// TwinCAT 3 PLC project LF_System_PLC
// ProgramVersion: 3.1.4026.20
// CompilerDefines: VISU_USEPROPERTYINFO
// libraries:
//   Tc2_Standard, * (Beckhoff Automation GmbH)
//   Tc2_System, * (Beckhoff Automation GmbH)
//   VisuSymbols, 4.5.0.0 (System)
// project tree:
//   / GlobalTextList.TcGTLO, PlcTask.TcTTO, Visualization Manager.TcVMO (not stored)
//   POUs/Extruder/ FB_System_FlaschenFullstand.TcPOU, FB_System_Fullstand.TcPOU
//   POUs/ FB_System_CNV.TcPOU (not stored), MAIN.TcPOU
//   POUs/Vereinzelung/ FB_SpeicherRohr.TcPOU, FB_System_Vereinzelung.TcPOU
//   VISUs/ Visualization.TcVIS
// (motion and I/O tree: see PLC project tempmodel)
// real-time tasks:
//   TASK PlcTask: cycle T#10ms, priority 21, ADS port 350
//   TASK PlcTask1: cycle T#10ms, priority 22, ADS port 351
//   TASK PlcTask2: cycle T#10ms, priority 20, ADS port 352
// variable links:
//   LF_System_PLC/LF_System_PLC Instance <-> NC-Task 1 SAF/Axes/BandAchse
//     PlcTask Inputs/MAIN.fIN_CnvPos <-> Outputs/ToPlc/ActPos
//   LF_System_PLC/LF_System_PLC Instance <-> PLC/PLC Instance
//     PlcTask Inputs/MAIN.bIn_LedGreen <-> PlcTask Outputs/IFC_HW.bAmpelGrun
//     PlcTask Inputs/MAIN.bIn_LedRot <-> PlcTask Outputs/IFC_HW.bAmpelRot
//     PlcTask Inputs/MAIN.bIn_LedYellow <-> PlcTask Outputs/IFC_HW.bAmpelGelb
//     PlcTask Inputs/MAIN.bIn_Schleuse1_L1 <-> PlcTask Outputs/IFC_HW.bR1AKT1
//     PlcTask Inputs/MAIN.bIn_Schleuse1_L2 <-> PlcTask Outputs/IFC_HW.bR2AKT1
//     PlcTask Inputs/MAIN.bIn_Schleuse2_L1 <-> PlcTask Outputs/IFC_HW.bR1AKT2
//     PlcTask Inputs/MAIN.bIn_Schleuse2_L2 <-> PlcTask Outputs/IFC_HW.bR2AKT2
//     PlcTask Outputs/MAIN.bEnable <-> PlcTask Inputs/IFC_HW.bEnable
//     PlcTask Outputs/MAIN.bExecute <-> PlcTask Inputs/IFC_HW.bExecute
//     PlcTask Outputs/MAIN.bOut_VereinzelungNS1 <-> PlcTask Inputs/IFC_HW.bEinzelSens3
//     PlcTask Outputs/MAIN.bOut_VereinzelungNS2 <-> PlcTask Inputs/IFC_HW.bEinzelSens2
//     PlcTask Outputs/MAIN.bOut_VereinzelungNS3 <-> PlcTask Inputs/IFC_HW.bEinzelSens1

CONFIGURATION LF_System_PLC
    RESOURCE PLC ON TwinCAT3
        TASK PlcTask(INTERVAL := T#10ms, PRIORITY := 22);
        PROGRAM MAIN WITH PlcTask : MAIN;
    END_RESOURCE
END_CONFIGURATION

// ---- POUs/MAIN.TcPOU
PROGRAM MAIN
VAR
// Systemeingangssignale (Stellsignale für Aktoren)
	bEnable AT%Q* : BOOL;
	bExecute AT%Q* : BOOL;
	// Status Lampe
	bIn_LedRot 		AT%I* : BOOL;
	bIn_LedYellow 	AT%I* : BOOL;
	bIn_LedGreen 	AT%I* : BOOL;
	// Vereinzelung 
	bIn_Schleuse1_L1 AT%I* : BOOL; // + Öffnen - Schließen
	bIn_Schleuse1_L2 AT%I* : BOOL; // + Schließen - Öffnen
	bIn_Schleuse2_L1 AT%I* : BOOL; // + Öffnen - Schließen
	bIn_Schleuse2_L2 AT%I* : BOOL; // + Schließen - Öffnen
	// Förderband
	fIN_CnvPos AT%I* : LREAL;
	bIN_Stopper1 AT%I* : BOOL;
	bIN_Stopper2 AT%I* : BOOL;
	bIN_Stopper3 AT%I* : BOOL;
	// Extruder
	fIN_ExtPos1 AT%I* : LREAL;
	fIN_ExtPos2 AT%I* : LREAL;
	fIN_ExtPos3 AT%I* : LREAL;
	
// Systemausgangssignale (Sensorsignale)
	//Vereinzelung
	bOut_VereinzelungNS1 AT%Q* : BOOL; // Flasche am Kopf
	bOut_VereinzelungNS2 AT%Q* : BOOL; // Flasche im Speicher
	bOut_VereinzelungNS3 AT%Q* : BOOL; // Flasche in Kammer
	//Förderband
	bOUT_CnvNS1 AT%Q* : BOOL;
	bOUT_CnvNS2 AT%Q* : BOOL;
	bOUT_CnvNS3 AT%Q* : BOOL;
	bOUT_CnvNS4 AT%Q* : BOOL;
	// Füllstandssensoren
	iOut_USS1 AT%Q* : UINT;
	iOut_USS2 AT%Q* : UINT;
	iOut_USS3 AT%Q* : UINT;
	
// System FB
	fbVereinzelung : FB_System_Vereinzelung;	
	fbCNV : FB_System_CNV;
	fbExt1 : FB_System_Fullstand;
	fbExt2 : FB_System_Fullstand;
	fbExt3 : FB_System_Fullstand;
	fbBottleLevel : FB_System_FlaschenFullstand;
	
// Hilfsvariablen
	bRefill1 : BOOL;
	bRefill2 : BOOL;
	bRefill3 : BOOL;
	bBottleDropped : BOOL;
	bBottleLeft : BOOL;
END_VAR

fbVereinzelung(
	bS1L1:= bIn_Schleuse1_L1, 
	bS1L2:= bIn_Schleuse1_L2, 
	bS2L1:= bIn_Schleuse2_L1, 
	bS2L2:= bIn_Schleuse2_L2,
	bNS1=> bOut_VereinzelungNS1, 
	bNS2=> bOut_VereinzelungNS2, 
	bNS3=> bOut_VereinzelungNS3,
	bBottleDropped => bBottleDropped);
	
fbCNV(
	fPos:= fIN_CnvPos, 
	bStopper1:= bIN_Stopper1, 
	bStopper2:= bIN_Stopper2, 
	bStopper3:= bIN_Stopper3, 
	bBottleDropped := bBottleDropped , 
	bNS1=> bOut_CnvNS1 , 
	bNS2=> bOut_CnvNS2 , 
	bNS3=> bOut_CnvNS3 , 
	bNS4=> bOut_CnvNS4,
	bBottleLeft => bBottleLeft);
	
fbExt1(bRefill:=bRefill1 , fPosExt:= fIN_ExtPos1, iOut=> iOut_USS1 );
fbExt2(bRefill:=bRefill2 , fPosExt:= fIN_ExtPos2, iOut=> iOut_USS2 );
fbExt3(bRefill:=bRefill3 , fPosExt:= fIN_ExtPos3, iOut=> iOut_USS3 );

fbBottleLevel(rFilling1 := fIN_ExtPos1, rFilling2 := fIN_ExtPos2 ,rFilling3 := fIN_ExtPos3,Reset:= bBottleLeft );

END_PROGRAM

// ---- POUs/Vereinzelung/FB_System_Vereinzelung.TcPOU
FUNCTION_BLOCK FB_System_Vereinzelung
VAR_INPUT
	bS1L1 : BOOL; // + Öffnen - Schließen
	bS1L2 : BOOL; // + Schließen - Öffnen
	bS2L1 : BOOL; // + Öffnen - Schließen
	bS2L2 : BOOL; // + Schließen - Öffnen
END_VAR
VAR_OUTPUT
	bNS1 : BOOL; // Flasche am Kopf
	bNS2 : BOOL; // Flasche im Speicher
	bNS3 : BOOL; // Flasche in Kammer
	bBottleDropped : BOOL;
END_VAR
VAR
	bS1open : BOOL;
	bS2open : BOOL;
	TimerS1 : Ton; // Schleusenbewegung (Schleuse1)
	TimerS2 : Ton; // Schleusenbewegung (Schleuse2)
	fbSpeicherRohr : FB_SpeicherRohr;
	nCaseS1 : UINT := 0;
	nCaseS2 : UINT := 0;
	bBefullen : BOOL;
	S1pos : INT;
	S2pos : INT;
END_VAR

TimerS1(PT := T#0.3S);
TimerS2(PT := T#0.3S);
fbSpeicherRohr(bFlascheBefullen:= bBefullen, bFlascheAuswurf := bS1open, bKammer := bNS3, bAuswurf => , aSpeicher => );

// Sensor in Speicher
bNS2 := fbSpeicherRohr.aSpeicher[0];
// Sensor in Kammer
IF fbSpeicherRohr.bAuswurf AND NOT bS2open THEN
	bNS3 := TRUE;
ELSIF bS2Open THEN
	bNS3 := FALSE;
END_IF

CASE nCaseS1 OF // Zustand S1
	0: // Schleuse geschlossen
	bS1open := FALSE;
	IF bS1L1 AND NOT bS1L2 THEN
		nCaseS1 := 1; // obere Schleuse öffnen
	END_IF
//------------------------------------------------	
	1: // obere Schleuse öffnen
	TimerS1.IN := TRUE;
	IF NOT bS1open THEN
		S1pos := S1pos - 1;
	END_IF
	IF TimerS1.Q THEN
		bS1open := TRUE;
	END_IF
	IF NOT bS1L1 AND bS1L2 THEN
		nCaseS1 := 2; // obere Schleuse schließen
		TimerS1.IN := FALSE;
	END_IF
//------------------------------------------------
	2: //obere Schleuse schließen
	TimerS1.IN := TRUE;
	IF bS1open THEN
		S1pos := S1pos + 1;
	END_IF
	IF timerS1.Q THEN
		bS1open := FALSE;
	END_IF
	IF bS1L1 AND NOT bS1L2 THEN
		nCaseS1 := 1; // obere Schleuse schließen
		TimerS1.IN := FALSE;
	END_IF
END_CASE

CASE nCaseS2 OF // Zustand S2
	0: // Schleuse geschlossen
	bS2open := FALSE;
	IF bS2L1 AND NOT bS2L2 THEN
		nCaseS2 := 1; // obere Schleuse öffnen
	END_IF
//------------------------------------------------	
	1: // untere Schleuse öffnen
	TimerS2.IN := TRUE;
	IF NOT bS2open THEN
		S2pos := S2pos - 1;
	END_IF
	IF TimerS2.Q THEN
		bS2open := TRUE;
	END_IF
	IF bS2open AND bNS3 THEN
		bBottleDropped := TRUE;
	END_IF
	IF NOT bS2L1 AND bS2L2 THEN
		nCaseS2 := 2; // untere Schleuse schließen
		TimerS2.IN := FALSE;
	END_IF
//------------------------------------------------
	2: //untere Schleuse schließen
	TimerS2.IN := TRUE;
	IF bS2open THEN
		S2pos := S2pos + 1;
	END_IF
	IF timerS2.Q THEN
		bS2open := FALSE;
		bBottleDropped := FALSE;
	END_IF
	IF bS2L1 AND NOT bS2L2 THEN
		nCaseS2 := 1; // untere Schleuse schließen
		TimerS2.IN := FALSE;
	END_IF
END_CASE

END_FUNCTION_BLOCK

// ---- POUs/Vereinzelung/FB_SpeicherRohr.TcPOU
FUNCTION_BLOCK FB_SpeicherRohr
VAR_INPUT
	bFlascheBefullen : BOOL; // Flasche soll in Speicher gelegt werden
	bFlascheAuswurf : BOOL; // Flasche soll in Kammer fallen
	bKammer : Bool;
END_VAR
VAR_OUTPUT
	bAuswurf : BOOL; // Flasche wurde ausgeworfen
	aSpeicher : ARRAY[0..3] OF BOOL := [TRUE,TRUE,TRUE,FALSE];
END_VAR
VAR
	rTrigBefullen : R_Trig;
	rTrigAuswurf : R_Trig;
	i : INT;
END_VAR

rTrigBefullen(CLK := bFlascheBefullen);
rTrigAuswurf(CLK := bFlascheAuswurf);

// Flaschenspeicher befüllen
IF rTrigBefullen.q AND NOT aSpeicher[3] THEN
	FOR i := 0 TO 3 DO
		IF NOT aSpeicher[i] THEN
			aSpeicher[i] := TRUE;
			EXIT;
		END_IF
	END_FOR
ELSIF rTrigBefullen.Q AND NOT aSpeicher[0] AND bFlascheAuswurf AND NOT bKammer THEN
	aSpeicher[0] := FALSE; 
	aSpeicher[1] := FALSE;
	aSpeicher[2] := FALSE;
	aSpeicher[3] := FALSE;
	bAuswurf := TRUE;
END_IF

IF rTrigAuswurf.q AND aSpeicher[0] THEN
	FOR i := 3 TO 0 BY -1 DO
		IF aSpeicher[i] THEN
			aSpeicher[i] := FALSE;
			EXIT;
		END_IF
	END_FOR
	bAuswurf := TRUE;
ELSE
	bAuswurf := FALSE; // Keine Flasche in Speicher
END_IF

END_FUNCTION_BLOCK

// ---- POUs/Extruder/FB_System_Fullstand.TcPOU
FUNCTION_BLOCK FB_System_Fullstand
VAR_INPUT
	bRefill : BOOL;
	fPosExt : LREAL;
END_VAR
VAR_OUTPUT
	iOut : UINT; // Fullstandssignal
END_VAR
VAR
	rPcntFillLevel : LREAL := 50.0; // Fullstand in Prozent
	iFillLevel : UINT;
	fPosExtAlt : LREAL;
	NotMoving : Bool;
END_VAR


// Auffüllen
IF bRefill THEN
	rPcntFillLevel := 100.0;
END_IF
// Füllstandsänderung durch Extruderbewegung
IF NOT notMoving THEN
	rPcntFillLevel := rPcntFillLevel - (fPosExt-fPosExtAlt)/360*0.5; // Füllstand - Grad/Umdrehung * 0,5% pro Umdrehung
END_IF

IF rPcntFillLevel < 0.0 THEN
	rPcntFillLevel := 0.0;
END_IF

iFillLevel := TO_UINT(rPcntFillLevel*1.7);

IF fPosExtAlt = fPosExt THEN
	NotMoving := TRUE;
ELSE
	NotMoving := FALSE;
END_IF

fPosExtAlt := fPosExt;

iOut := to_UINT(-65536/100 * rPcntFillLevel + 65536);

END_FUNCTION_BLOCK

// ---- POUs/Extruder/FB_System_FlaschenFullstand.TcPOU
FUNCTION_BLOCK FB_System_FlaschenFullstand
VAR_INPUT
	rFilling1 : LREAL;
	rFilling2 : LREAL;
	rFilling3 : LREAL;
	Reset : BOOL;
END_VAR
VAR_OUTPUT
END_VAR
VAR
	rPcntFillLevel : LREAL;
	rFilling1Alt : LREAL;
	rFilling2Alt : LREAL;
	rFilling3Alt : LREAL;
	iFillLevel1 : UINT;
	iFillLevel2 : UINT;
	iFillLevel3 : UINT;
END_VAR

IF Reset THEN
	rPcntFillLevel := 0.0;
	iFillLevel1 := 0;
	iFillLevel2 := 0;
	iFillLevel3 := 0;
END_IF

IF rFilling1 <> rFilling1Alt THEN 
	rPcntFillLevel := rPcntFillLevel + (rFilling1 - rFilling1Alt)/360*7;
	iFillLevel1 := TO_UINT(rPcntFillLevel * 0.25);
ELSIF rFilling2 <> rFilling2Alt THEN
	rPcntFillLevel := rPcntFillLevel + (rFilling2 - rFilling2Alt)/360*7;
	iFillLevel2 := TO_UINT(rPcntFillLevel * 0.25)-iFillLevel1;
ELSIF rFilling3 <> rFilling3Alt THEN
	rPcntFillLevel := rPcntFillLevel + (rFilling3 - rFilling3Alt)/360*7;
	iFillLevel3 := TO_UINT(rPcntFillLevel * 0.25)- iFillLevel2-iFillLevel1;
END_IF

rFilling1Alt := rFilling1;
rFilling2Alt := rFilling2;
rFilling3Alt := rFilling3;

IF rPcntFillLevel > 100 THEN
	rPcntFillLevel := 100.0;
END_IF

END_FUNCTION_BLOCK

// ---- GlobalTextList.TcGTLO
TEXTLIST GlobalTextList
  477 = 'Befüllen'
  647 = 'Enable'
  925 = 'Execute'
END_TEXTLIST

// ---- VISUs/Visualization.TcVIS
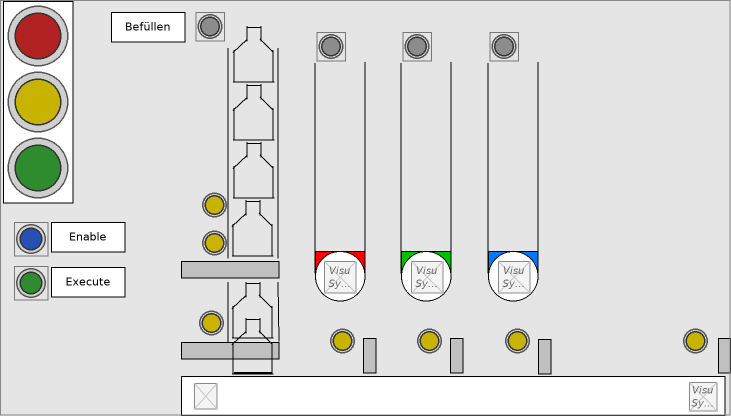
VISUALIZATION Visualization  // 731x416
    Rectangle (315,251 50x24)
        p2773130477: - MAIN.fbExt1.iFillLevel
    Lamp1 (200,190 29x30), variable: MAIN.bOut_VereinzelungNS1, style: Lamp-Lamp1-Yellow
    Lamp1 (200,228 29x30), variable: MAIN.bOut_VereinzelungNS2, style: Lamp-Lamp1-Yellow
    Lamp1 (197,308 29x30), variable: MAIN.bOut_VereinzelungNS3, style: Lamp-Lamp1-Yellow
    Group (3,1 70x202)
        Rectangle (0,0 70x202)
        Lamp1 (0,0 70x70), variable: MAIN.bIn_LedRot, style: Lamp-Lamp1-Red
        Lamp1 (0,66 70x70), variable: MAIN.bIn_LedYellow, style: Lamp-Lamp1-Yellow
        Lamp1 (0,132 70x70), variable: MAIN.bIn_LedGreen, style: Lamp-Lamp1-Green
    Line (228,258) (228,48)
    Line (278,258) (278,48)
    Line (279,341) (278,282)
    Line (228,342) (228,282)
    Rectangle (181,261 98x17)
        p3528305787: MAIN.fbVereinzelung.S1pos
        p874137650: MAIN.fbVereinzelung.S1pos
    Rectangle (181,342 98x17)
        p3528305787: MAIN.fbVereinzelung.S2pos
        p874137650: MAIN.fbVereinzelung.S2pos
    PushSwitch (12,222 38x34), variable: MAIN.bEnable, behaviour: TOGGLE, style: Switch-PushSwitch-Blue
    PushSwitch (12,266 38x34), variable: MAIN.bExecute, behaviour: TAP, style: Switch-PushSwitch-Green
    Rectangle (51,222 74x30), "Enable"
    Rectangle (51,267 74x30), "Execute"
    Group (232,200 41x57), invisible if: not MAIN.fbVereinzelung.fbSpeicherRohr.aSpeicher[0]
        Line (1,56) (1,24)
        Line (40,55) (40,24)
        Line (41,56) (0,56)
        Line (0,26) (14,13)
        Line (40,26) (27,13)
        Line (14,15) (14,0)
        Line (28,15) (28,0)
        Line (14,1) (28,1)
    Group (233,142 41x57), invisible if: Not MAIN.fbVereinzelung.fbSpeicherRohr.aSpeicher[1]
        Line (1,56) (1,24)
        Line (40,55) (40,24)
        Line (41,56) (0,56)
        Line (0,26) (14,13)
        Line (40,26) (27,13)
        Line (14,15) (14,0)
        Line (28,15) (28,0)
        Line (14,1) (28,1)
    Group (232,282 41x57), invisible if: not MAIN.bOut_VereinzelungNS3
        Line (1,56) (1,24)
        Line (40,55) (40,24)
        Line (41,56) (0,56)
        Line (0,26) (14,13)
        Line (40,26) (27,13)
        Line (14,15) (14,0)
        Line (28,15) (28,0)
        Line (14,1) (28,1)
    Group (233,84 41x57), invisible if: Not MAIN.fbVereinzelung.fbSpeicherRohr.aSpeicher[2]
        Line (1,56) (1,24)
        Line (40,55) (40,24)
        Line (41,56) (0,56)
        Line (0,26) (14,13)
        Line (40,26) (27,13)
        Line (14,15) (14,0)
        Line (28,15) (28,0)
        Line (14,1) (28,1)
    Group (233,26 41x57), invisible if: Not MAIN.fbVereinzelung.fbSpeicherRohr.aSpeicher[3]
        Line (1,56) (1,24)
        Line (40,55) (40,24)
        Line (41,56) (0,56)
        Line (0,26) (14,13)
        Line (40,26) (27,13)
        Line (14,15) (14,0)
        Line (28,15) (28,0)
        Line (14,1) (28,1)
    PushSwitch (194,12 32x29), variable: MAIN.fbVereinzelung.bBefullen, behaviour: TAP, style: Switch-PushSwitch-Gray
    RoundedRectangle (181,376 544x40)
    Lamp1 (328,326 29x30), variable: MAIN.bOUT_CnvNS1, style: Lamp-Lamp1-Yellow
    Lamp1 (503,326 29x30), variable: MAIN.bOUT_CnvNS3, style: Lamp-Lamp1-Yellow
    Lamp1 (415,326 29x30), variable: MAIN.bOUT_CnvNS2, style: Lamp-Lamp1-Yellow
    Lamp1 (681,326 29x30), variable: MAIN.bOUT_CnvNS4, style: Lamp-Lamp1-Yellow
    Group (232,318 41x57), invisible if: not MAIN.fbCNV.bBottleOnCNV
        p3560616238: MAIN.fbCNV.iBottlePos
        Line (1,56) (1,24)
        Line (40,55) (40,24)
        Line (41,56) (0,56)
        Line (0,26) (14,13)
        Line (40,26) (27,13)
        Line (14,15) (14,0)
        Line (28,15) (28,0)
        Line (14,1) (28,1)
    Rectangle (363,338 13x35), invisible if: MAIN.bIN_Stopper1
    Rectangle (450,338 13x35), invisible if: MAIN.bIN_Stopper2
    Rectangle (538,339 13x35), invisible if: MAIN.bIN_Stopper3
    Rectangle (718,338 13x35)
    Image (194,383 23x26), invisible if: not MAIN.fbCNV.bCNVisMoving, image: VisuSymbols.Symbols.ArrowHalfRightUp
    Image (689,382 28x29), invisible if: not MAIN.fbCNV.bCNVisMoving, image: VisuSymbols.Symbols.ArrowHalfRightDown
    Rectangle (111,12 74x30), "Befüllen"
    Ellipse (315,251 50x50)
    Line (315,273) (315,63)
    Line (365,272) (365,62)
    Rectangle (401,251 50x24)
        p2773130477: - MAIN.fbExt2.iFillLevel
    Ellipse (401,251 50x50)
    Line (401,273) (401,63)
    Line (451,272) (451,62)
    Rectangle (488,251 50x24)
        p2773130477: - MAIN.fbExt3.iFillLevel
    Ellipse (488,251 50x50)
    Line (488,273) (488,63)
    Line (538,272) (538,62)
    PushSwitch (315,32 32x29), variable: MAIN.bRefill1, behaviour: TAP, style: Switch-PushSwitch-Gray
    PushSwitch (401,32 32x29), variable: MAIN.bRefill2, behaviour: TAP, style: Switch-PushSwitch-Gray
    PushSwitch (488,32 32x29), variable: MAIN.bRefill3, behaviour: TAP, style: Switch-PushSwitch-Gray
    Image (324,261 32x32), invisible if: MAIN.fbExt1.NotMoving, image: VisuSymbols.Symbols.ArrowCircle2RightRightLeft
    Image (411,261 32x32), invisible if: MAIN.fbExt2.NotMoving, image: VisuSymbols.Symbols.ArrowCircle2RightRightLeft
    Image (498,261 32x32), invisible if: MAIN.fbExt3.NotMoving, image: VisuSymbols.Symbols.ArrowCircle2RightRightLeft
    Rectangle (234,372 38x1), invisible if: not MAIN.fbCNV.bBottleOnCNV
        p2773130477: - MAIN.fbBottleLevel.iFillLevel3 - MAIN.fbBottleLevel.iFillLevel1 - MAIN.fbBottleLevel.iFillLevel2
        p3560616238: MAIN.fbCNV.iBottlePos
        p1126004900: - MAIN.fbBottleLevel.iFillLevel1 - MAIN.fbBottleLevel.iFillLevel2
    Rectangle (234,372 38x1), invisible if: not MAIN.fbCNV.bBottleOnCNV
        p2773130477: - MAIN.fbBottleLevel.iFillLevel2 - MAIN.fbBottleLevel.iFillLevel1
        p3560616238: MAIN.fbCNV.iBottlePos
        p1126004900: - MAIN.fbBottleLevel.iFillLevel1
    Rectangle (234,372 38x1), invisible if: not MAIN.fbCNV.bBottleOnCNV
        p2773130477: - MAIN.fbBottleLevel.iFillLevel1
        p3560616238: MAIN.fbCNV.iBottlePos
END_VISUALIZATION
